# EPICS alarm handler configuration: mps_database/bareTest/alarms/areas/mpln_undh_mp09.alhConfig
GROUP NULL MPLN:UNDH:MP09:1
$ALIAS MPS Link Node 144
$GUIDANCE
LTUH MPS
   Group Name: MPLN:UNDH:MP09:1
   Summary PV:  MPLN:UNDH:MP09:1:STATSUMY
$END
CHANNEL  MPLN:UNDH:MP09:1    MPLN:UNDH:MP09:1:MPS_EN_RBV		-----
CHANNEL  MPLN:UNDH:MP09:1    MPLN:UNDH:MP09:1:LC1_MODE_RBV		-----
